FUNCTION alg_a_HledQ2 : BOOL
VAR_INPUT
	state: STATE;
END_VAR

alg_a_HledQ2 := FALSE;

END_FUNCTION

(* stored: Version 1.1.0.1, ProductVersion 3.1.4022.18
   POU alg_a_HledQ2: Id {ca660977-cbc5-4857-b822-ee8bc483505e}, SpecialFunc None *)
